(* CoDeSys 2.3.9.50 project: 3E.pr6 *)
(* Libraries: STANDARD.LB6 5.6.98 12:03:02 *)

(* POU MAIN, LD *)
PROGRAM MAIN
VAR
	AlarmStart AT %IX0.0: BOOL;
	lightA AT %QX0.1: BOOL;
	lightB AT %QX0.2: BOOL;
	lightC AT %QX0.3: BOOL;
	lightD AT %QX0.4: BOOL;
	t1: TON;
	t2: TON;
END_VAR
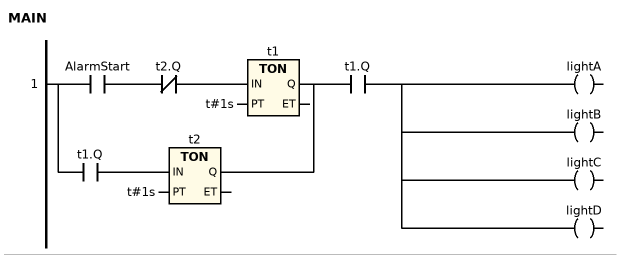
_LD_ (* Ladder Diagram *)
NETWORK 1
	{ [AlarmStart] - [/t2.Q] - t1:TON(IN: *, PT: t#1s) | [t1.Q] - t2:TON(IN: *, PT: t#1s) } - [t1.Q] --- (lightA) (lightB) (lightC) (lightD)
_END_LD_
(* the same logic as Structured Text *)
(* Network 1 *)
t1(IN := AlarmStart AND NOT t2.Q, PT := t#1s);
t2(IN := t1.Q, PT := t#1s);
lightA := (t1.Q OR t2.Q) AND t1.Q;
lightB := lightA;
lightC := lightA;
lightD := lightA;
END_PROGRAM
